TYPE UDT_LogHandlerConfig :
STRUCT
	pLogHandler 		: POINTER TO FB_LogHandlerBase := 0;
	eMinimumLogLevel 	: E_LogLevel := E_LogLevel.TRACE;
END_STRUCT
END_TYPE

(* stored: Version 1.1.0.1, ProductVersion 3.1.4024.11
   DUT UDT_LogHandlerConfig: Id {5f749529-f5f6-0a93-3e9e-0af39aea1f0e} *)
